VAR_GLOBAL
	PositionerIsClamped	:	BOOL;
	PositionerIsRaised	:	BOOL;
	PositionerClamp	:	BOOL;
	PositionerRaise	:	BOOL;
END_VAR

(* stored: Version 1.1.0.1
   GVL PositioningBar: Id {93bed95a-dcb1-49b3-a7bf-8028c1278755} *)
